(* Logix 5000 project; controller Uidaho_Factory vendor 1 type 14 code 165 rev 38.11; software revision 38.00; part 2 of 2 *)
(* tags used below, declared in another part *)
   StepTimers : TIMER[20];
   VGR_HBW_Horizontal : DINT;   // The horizontal Encoder value for interfacing with HBW
   VGR_HBW_Rotate : DINT;
   VGR_HBW_Vertical : DINT;   // The Vertical Encoder value for interfacing with the HBW
   VGR_Horizontal_Target : DINT;
   VGR_Move_Horizontal : DINT;   // The horizontal encoder value for movement
   VGR_Move_Vertical : DINT;   // The vertical encoder value for movement
   VGR_MPO_Horizontal : DINT;   // The Horizontal encoderr value for interfacing with MPO
   VGR_MPO_Rotate : DINT;
   VGR_MPO_Vertical : DINT;   // The vertical encoder value for interfacing with MPO
   VGR_Rotation_Target : DINT;
   VGR_start : DINT;
   VGR_Step : DINT;
   VGR_Vertical_Target : DINT;
   Encoder_Counters_1X : COUNTER[10];
   Encoder_Output_Bits_VGR : DINT[2];
   Encoder_Storage_Bits_VGR : DINT[2];
(* MainProgram, continued *)

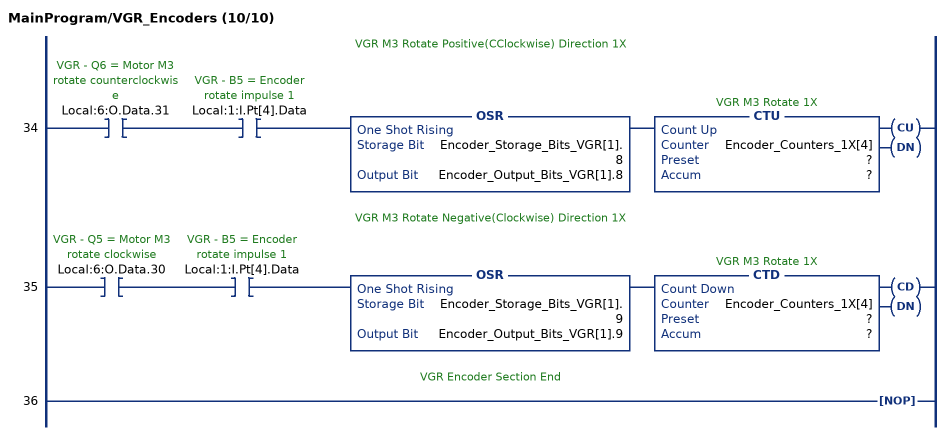
   [picture p24: MainProgram/VGR_Encoders rungs 34-36]
   // VGR M3 Rotate Positive(CClockwise) Direction 1X
   34: XIC(Local:6:O.Data.31)XIC(Local:1:I.Pt[4].Data)OSR(Encoder_Storage_Bits_VGR[1].8,Encoder_Output_Bits_VGR[1].8)CTU(Encoder_Counters_1X[4],?,?);
   // VGR M3 Rotate Negative(Clockwise) Direction 1X
   35: XIC(Local:6:O.Data.30)XIC(Local:1:I.Pt[4].Data)OSR(Encoder_Storage_Bits_VGR[1].9,Encoder_Output_Bits_VGR[1].9)CTD(Encoder_Counters_1X[4],?,?);
   // VGR Encoder Section End
   36: NOP();
END_ROUTINE

ROUTINE VGR_Sequencer   (* ladder *)
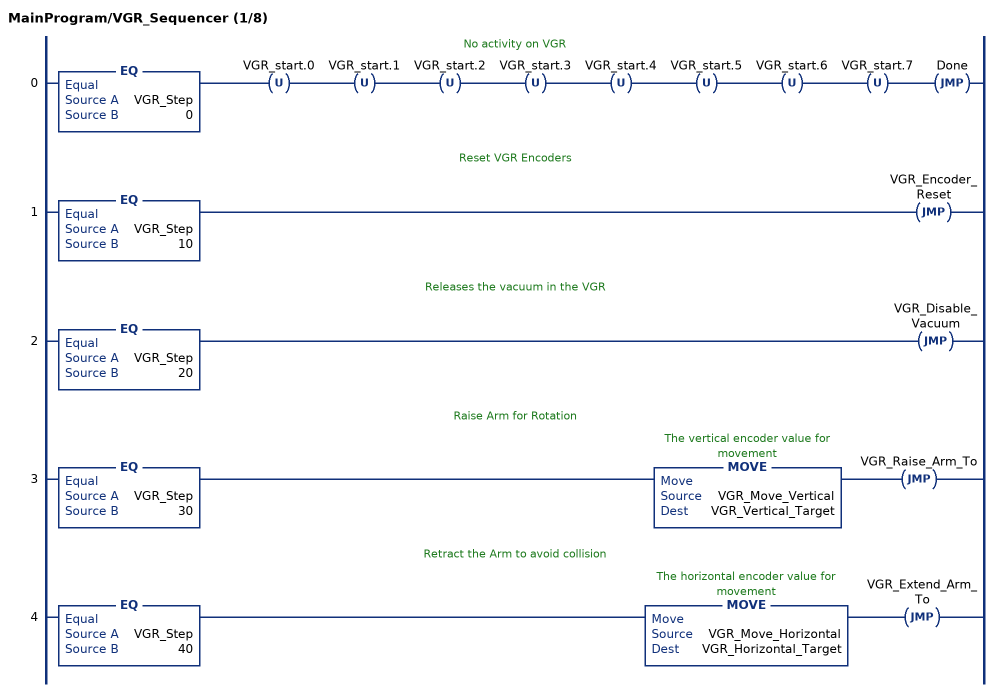
   // No activity on VGR
   0: EQ(VGR_Step,0)OTU(VGR_start.0)OTU(VGR_start.1)OTU(VGR_start.2)OTU(VGR_start.3)OTU(VGR_start.4)OTU(VGR_start.5)OTU(VGR_start.6)OTU(VGR_start.7)JMP(Done);
   // Reset VGR Encoders
   1: EQ(VGR_Step,10)JMP(VGR_Encoder_Reset);
   // Releases the vacuum in the VGR
   2: EQ(VGR_Step,20)JMP(VGR_Disable_Vacuum);
   // Raise Arm for Rotation
   3: EQ(VGR_Step,30)MOVE(VGR_Move_Vertical,VGR_Vertical_Target)JMP(VGR_Raise_Arm_To);
   // Retract the Arm to avoid collision
   4: EQ(VGR_Step,40)MOVE(VGR_Move_Horizontal,VGR_Horizontal_Target)JMP(VGR_Extend_Arm_To);
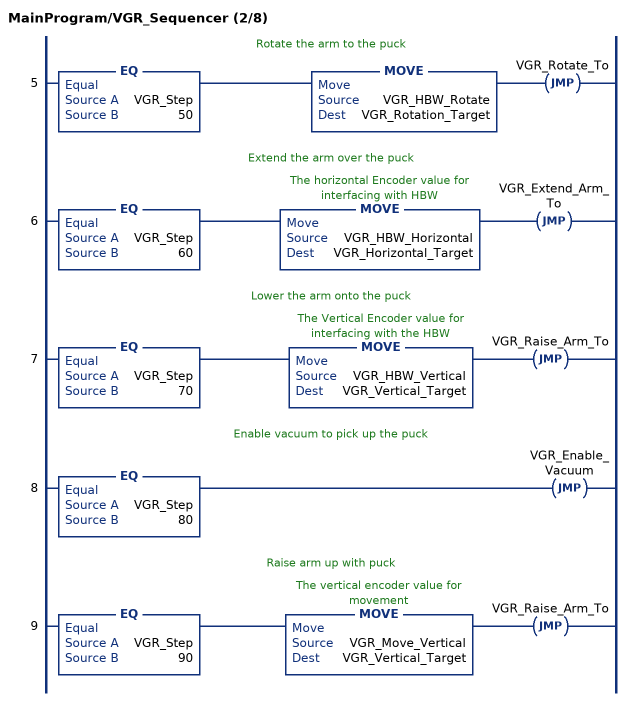
   // Rotate the arm to the puck
   5: EQ(VGR_Step,50)MOVE(VGR_HBW_Rotate,VGR_Rotation_Target)JMP(VGR_Rotate_To);
   // Extend the arm over the puck
   6: EQ(VGR_Step,60)MOVE(VGR_HBW_Horizontal,VGR_Horizontal_Target)JMP(VGR_Extend_Arm_To);
   // Lower the arm onto the puck
   7: EQ(VGR_Step,70)MOVE(VGR_HBW_Vertical,VGR_Vertical_Target)JMP(VGR_Raise_Arm_To);
   // Enable vacuum to pick up the puck
   8: EQ(VGR_Step,80)JMP(VGR_Enable_Vacuum);
   // Raise arm up with puck
   9: EQ(VGR_Step,90)MOVE(VGR_Move_Vertical,VGR_Vertical_Target)JMP(VGR_Raise_Arm_To);
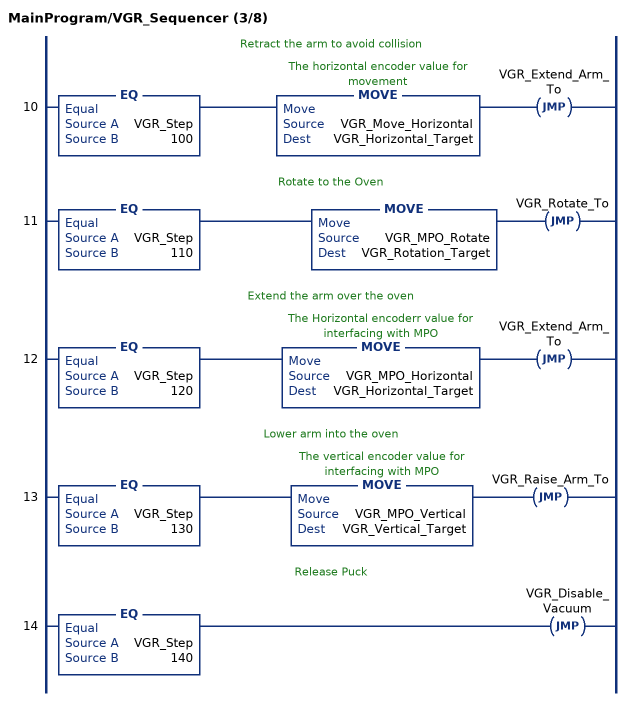
   // Retract the arm to avoid collision
   10: EQ(VGR_Step,100)MOVE(VGR_Move_Horizontal,VGR_Horizontal_Target)JMP(VGR_Extend_Arm_To);
   // Rotate to the Oven
   11: EQ(VGR_Step,110)MOVE(VGR_MPO_Rotate,VGR_Rotation_Target)JMP(VGR_Rotate_To);
   // Extend the arm over the oven
   12: EQ(VGR_Step,120)MOVE(VGR_MPO_Horizontal,VGR_Horizontal_Target)JMP(VGR_Extend_Arm_To);
   // Lower arm into the oven
   13: EQ(VGR_Step,130)MOVE(VGR_MPO_Vertical,VGR_Vertical_Target)JMP(VGR_Raise_Arm_To);
   // Release Puck
   14: EQ(VGR_Step,140)JMP(VGR_Disable_Vacuum);
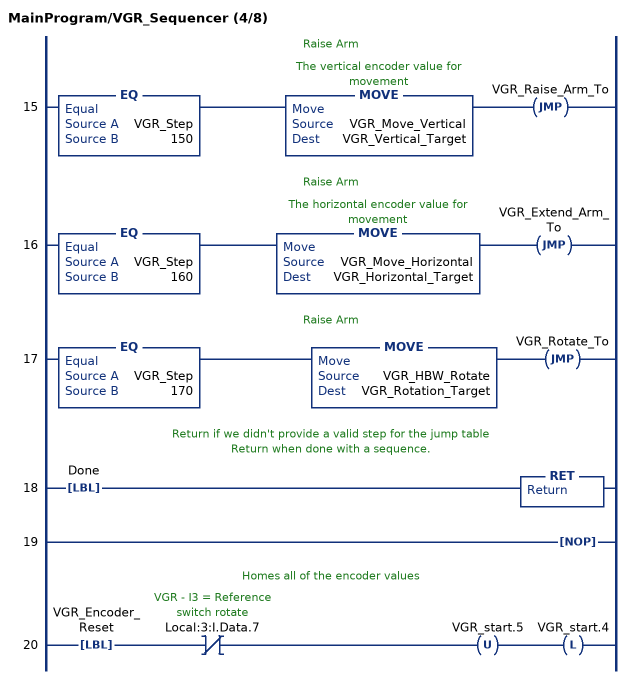
   // Raise Arm
   15: EQ(VGR_Step,150)MOVE(VGR_Move_Vertical,VGR_Vertical_Target)JMP(VGR_Raise_Arm_To);
   // Raise Arm
   16: EQ(VGR_Step,160)MOVE(VGR_Move_Horizontal,VGR_Horizontal_Target)JMP(VGR_Extend_Arm_To);
   // Raise Arm
   17: EQ(VGR_Step,170)MOVE(VGR_HBW_Rotate,VGR_Rotation_Target)JMP(VGR_Rotate_To);
   // Return if we didn't provide a valid step for the jump table
   // Return when done with a sequence.
   18: LBL(Done)RET();
   19: NOP();
   // Homes all of the encoder values
   20: LBL(VGR_Encoder_Reset)XIO(Local:3:I.Data.7)OTU(VGR_start.5)OTL(VGR_start.4);
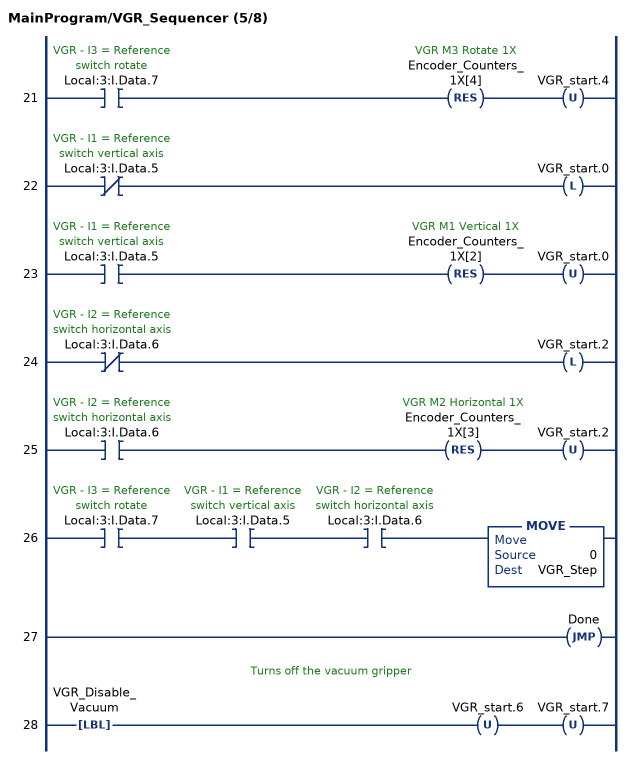
   21: XIC(Local:3:I.Data.7)RES(Encoder_Counters_1X[4])OTU(VGR_start.4);
   22: XIO(Local:3:I.Data.5)OTL(VGR_start.0);
   23: XIC(Local:3:I.Data.5)RES(Encoder_Counters_1X[2])OTU(VGR_start.0);
   24: XIO(Local:3:I.Data.6)OTL(VGR_start.2);
   25: XIC(Local:3:I.Data.6)RES(Encoder_Counters_1X[3])OTU(VGR_start.2);
   26: XIC(Local:3:I.Data.7)XIC(Local:3:I.Data.5)XIC(Local:3:I.Data.6)MOVE(0,VGR_Step);
   27: JMP(Done);
   // Turns off the vacuum gripper
   28: LBL(VGR_Disable_Vacuum)OTU(VGR_start.6)OTU(VGR_start.7);
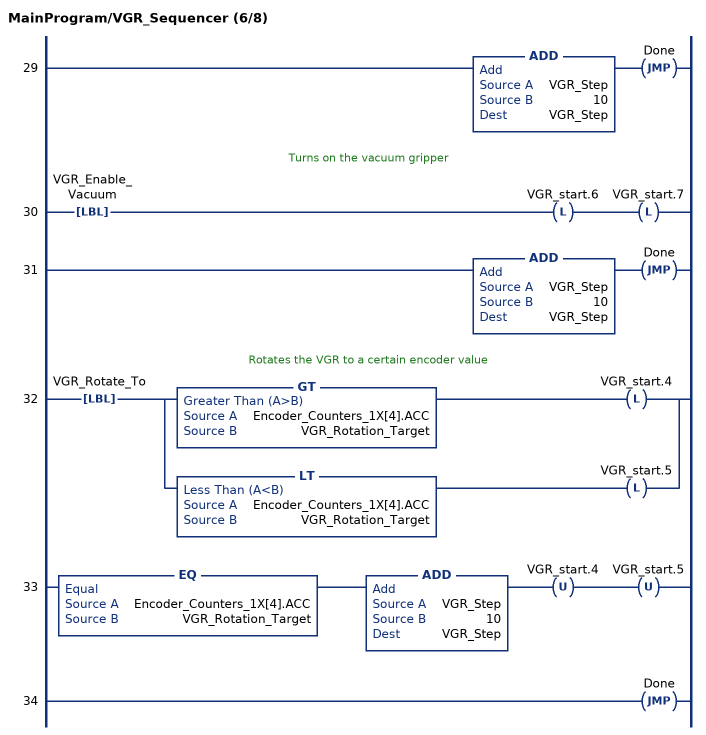
   29: ADD(VGR_Step,10,VGR_Step)JMP(Done);
   // Turns on the vacuum gripper
   30: LBL(VGR_Enable_Vacuum)OTL(VGR_start.6)OTL(VGR_start.7);
   31: ADD(VGR_Step,10,VGR_Step)JMP(Done);
   // Rotates the VGR to a certain encoder value
   32: LBL(VGR_Rotate_To)[GT(Encoder_Counters_1X[4].ACC,VGR_Rotation_Target) OTL(VGR_start.4) ,LT(Encoder_Counters_1X[4].ACC,VGR_Rotation_Target) OTL(VGR_start.5) ];
   33: EQ(Encoder_Counters_1X[4].ACC,VGR_Rotation_Target)ADD(VGR_Step,10,VGR_Step)OTU(VGR_start.4)OTU(VGR_start.5);
   34: JMP(Done);
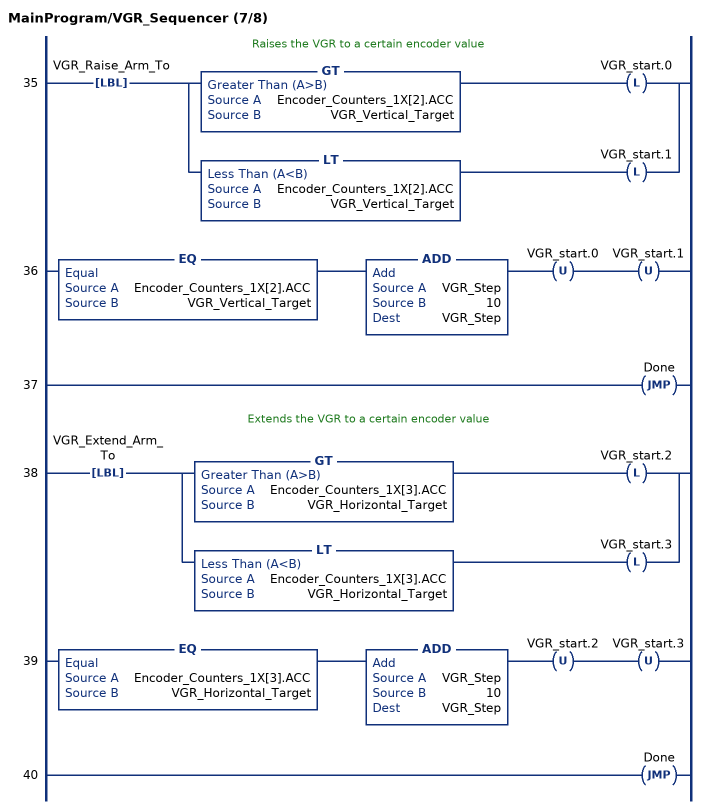
   // Raises the VGR to a certain encoder value
   35: LBL(VGR_Raise_Arm_To)[GT(Encoder_Counters_1X[2].ACC,VGR_Vertical_Target) OTL(VGR_start.0) ,LT(Encoder_Counters_1X[2].ACC,VGR_Vertical_Target) OTL(VGR_start.1) ];
   36: EQ(Encoder_Counters_1X[2].ACC,VGR_Vertical_Target)ADD(VGR_Step,10,VGR_Step)OTU(VGR_start.0)OTU(VGR_start.1);
   37: JMP(Done);
   // Extends the VGR to a certain encoder value
   38: LBL(VGR_Extend_Arm_To)[GT(Encoder_Counters_1X[3].ACC,VGR_Horizontal_Target) OTL(VGR_start.2) ,LT(Encoder_Counters_1X[3].ACC,VGR_Horizontal_Target) OTL(VGR_start.3) ];
   39: EQ(Encoder_Counters_1X[3].ACC,VGR_Horizontal_Target)ADD(VGR_Step,10,VGR_Step)OTU(VGR_start.2)OTU(VGR_start.3);
   40: JMP(Done);
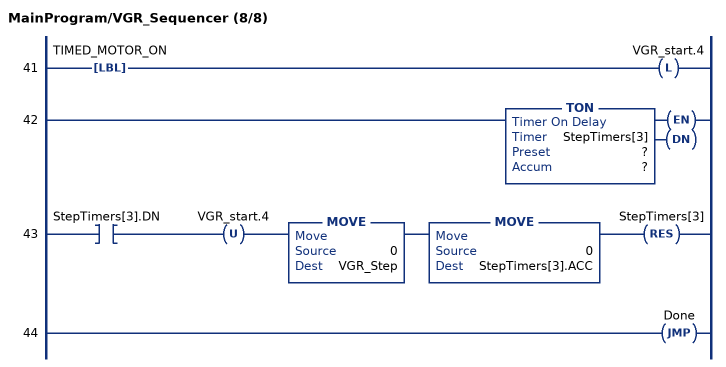
   41: LBL(TIMED_MOTOR_ON)OTL(VGR_start.4);
   42: TON(StepTimers[3],?,?);
   43: XIC(StepTimers[3].DN)OTU(VGR_start.4)MOVE(0,VGR_Step)MOVE(0,StepTimers[3].ACC)RES(StepTimers[3]);
   44: JMP(Done);
END_ROUTINE
END_PROGRAM
